FUNCTION_BLOCK SPLIT_AL_INTO_AQ (* this Function splits the 32 AQ (QUARTER) adapters from a AL (LWORD) *)
  (* Standard: 61499-2; Description: Copyright (c) 2026 Meisterschulen am Ostbahnhof SPDX-License-Identifier: EPL-2.0 *)
  (* Version 1.0, 2026-05-16, Franz Höpfinger, Meisterschulen am Ostbahnhof, initial API and implementation and/or initial documentation *)
  PACKAGE adapter::splitting;
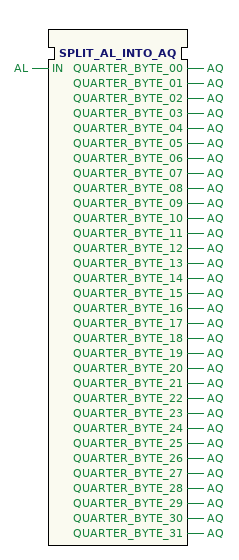
  SOCKETS
    IN : adapter::types::unidirectional::AL; (* LWORD Input *)
  END_SOCKETS
  PLUGS
    QUARTER_BYTE_00 : adapter::types::unidirectional::AQ; (* Quarter 0 *)
    QUARTER_BYTE_01 : adapter::types::unidirectional::AQ; (* Quarter 1 *)
    QUARTER_BYTE_02 : adapter::types::unidirectional::AQ; (* Quarter 2 *)
    QUARTER_BYTE_03 : adapter::types::unidirectional::AQ; (* Quarter 3 *)
    QUARTER_BYTE_04 : adapter::types::unidirectional::AQ; (* Quarter 4 *)
    QUARTER_BYTE_05 : adapter::types::unidirectional::AQ; (* Quarter 5 *)
    QUARTER_BYTE_06 : adapter::types::unidirectional::AQ; (* Quarter 6 *)
    QUARTER_BYTE_07 : adapter::types::unidirectional::AQ; (* Quarter 7 *)
    QUARTER_BYTE_08 : adapter::types::unidirectional::AQ; (* Quarter 8 *)
    QUARTER_BYTE_09 : adapter::types::unidirectional::AQ; (* Quarter 9 *)
    QUARTER_BYTE_10 : adapter::types::unidirectional::AQ; (* Quarter 10 *)
    QUARTER_BYTE_11 : adapter::types::unidirectional::AQ; (* Quarter 11 *)
    QUARTER_BYTE_12 : adapter::types::unidirectional::AQ; (* Quarter 12 *)
    QUARTER_BYTE_13 : adapter::types::unidirectional::AQ; (* Quarter 13 *)
    QUARTER_BYTE_14 : adapter::types::unidirectional::AQ; (* Quarter 14 *)
    QUARTER_BYTE_15 : adapter::types::unidirectional::AQ; (* Quarter 15 *)
    QUARTER_BYTE_16 : adapter::types::unidirectional::AQ; (* Quarter 16 *)
    QUARTER_BYTE_17 : adapter::types::unidirectional::AQ; (* Quarter 17 *)
    QUARTER_BYTE_18 : adapter::types::unidirectional::AQ; (* Quarter 18 *)
    QUARTER_BYTE_19 : adapter::types::unidirectional::AQ; (* Quarter 19 *)
    QUARTER_BYTE_20 : adapter::types::unidirectional::AQ; (* Quarter 20 *)
    QUARTER_BYTE_21 : adapter::types::unidirectional::AQ; (* Quarter 21 *)
    QUARTER_BYTE_22 : adapter::types::unidirectional::AQ; (* Quarter 22 *)
    QUARTER_BYTE_23 : adapter::types::unidirectional::AQ; (* Quarter 23 *)
    QUARTER_BYTE_24 : adapter::types::unidirectional::AQ; (* Quarter 24 *)
    QUARTER_BYTE_25 : adapter::types::unidirectional::AQ; (* Quarter 25 *)
    QUARTER_BYTE_26 : adapter::types::unidirectional::AQ; (* Quarter 26 *)
    QUARTER_BYTE_27 : adapter::types::unidirectional::AQ; (* Quarter 27 *)
    QUARTER_BYTE_28 : adapter::types::unidirectional::AQ; (* Quarter 28 *)
    QUARTER_BYTE_29 : adapter::types::unidirectional::AQ; (* Quarter 29 *)
    QUARTER_BYTE_30 : adapter::types::unidirectional::AQ; (* Quarter 30 *)
    QUARTER_BYTE_31 : adapter::types::unidirectional::AQ; (* Quarter 31 *)
  END_PLUGS
  FBS
    E_D_FF_ANY_00 : iec61499::events::E_D_FF_ANY;
    E_D_FF_ANY_01 : iec61499::events::E_D_FF_ANY;
    E_D_FF_ANY_02 : iec61499::events::E_D_FF_ANY;
    E_D_FF_ANY_03 : iec61499::events::E_D_FF_ANY;
    E_D_FF_ANY_04 : iec61499::events::E_D_FF_ANY;
    E_D_FF_ANY_05 : iec61499::events::E_D_FF_ANY;
    E_D_FF_ANY_06 : iec61499::events::E_D_FF_ANY;
    E_D_FF_ANY_07 : iec61499::events::E_D_FF_ANY;
    E_D_FF_ANY_08 : iec61499::events::E_D_FF_ANY;
    E_D_FF_ANY_09 : iec61499::events::E_D_FF_ANY;
    E_D_FF_ANY_10 : iec61499::events::E_D_FF_ANY;
    E_D_FF_ANY_11 : iec61499::events::E_D_FF_ANY;
    E_D_FF_ANY_12 : iec61499::events::E_D_FF_ANY;
    E_D_FF_ANY_13 : iec61499::events::E_D_FF_ANY;
    E_D_FF_ANY_14 : iec61499::events::E_D_FF_ANY;
    E_D_FF_ANY_15 : iec61499::events::E_D_FF_ANY;
    E_D_FF_ANY_16 : iec61499::events::E_D_FF_ANY;
    E_D_FF_ANY_17 : iec61499::events::E_D_FF_ANY;
    E_D_FF_ANY_18 : iec61499::events::E_D_FF_ANY;
    E_D_FF_ANY_19 : iec61499::events::E_D_FF_ANY;
    E_D_FF_ANY_20 : iec61499::events::E_D_FF_ANY;
    E_D_FF_ANY_21 : iec61499::events::E_D_FF_ANY;
    E_D_FF_ANY_22 : iec61499::events::E_D_FF_ANY;
    E_D_FF_ANY_23 : iec61499::events::E_D_FF_ANY;
    E_D_FF_ANY_24 : iec61499::events::E_D_FF_ANY;
    E_D_FF_ANY_25 : iec61499::events::E_D_FF_ANY;
    E_D_FF_ANY_26 : iec61499::events::E_D_FF_ANY;
    E_D_FF_ANY_27 : iec61499::events::E_D_FF_ANY;
    E_D_FF_ANY_28 : iec61499::events::E_D_FF_ANY;
    E_D_FF_ANY_29 : iec61499::events::E_D_FF_ANY;
    E_D_FF_ANY_30 : iec61499::events::E_D_FF_ANY;
    E_D_FF_ANY_31 : iec61499::events::E_D_FF_ANY;
    SPLIT_LWORD_INTO_QUARTERS : eclipse4diac::utils::splitting::SPLIT_LWORD_INTO_QUARTERS;
  END_FBS
  EVENT_CONNECTIONS
    IN.E1 TO SPLIT_LWORD_INTO_QUARTERS.REQ;
    SPLIT_LWORD_INTO_QUARTERS.CNF TO E_D_FF_ANY_00.CLK;
    SPLIT_LWORD_INTO_QUARTERS.CNF TO E_D_FF_ANY_01.CLK;
    SPLIT_LWORD_INTO_QUARTERS.CNF TO E_D_FF_ANY_02.CLK;
    SPLIT_LWORD_INTO_QUARTERS.CNF TO E_D_FF_ANY_03.CLK;
    SPLIT_LWORD_INTO_QUARTERS.CNF TO E_D_FF_ANY_04.CLK;
    SPLIT_LWORD_INTO_QUARTERS.CNF TO E_D_FF_ANY_05.CLK;
    SPLIT_LWORD_INTO_QUARTERS.CNF TO E_D_FF_ANY_06.CLK;
    SPLIT_LWORD_INTO_QUARTERS.CNF TO E_D_FF_ANY_07.CLK;
    SPLIT_LWORD_INTO_QUARTERS.CNF TO E_D_FF_ANY_08.CLK;
    SPLIT_LWORD_INTO_QUARTERS.CNF TO E_D_FF_ANY_09.CLK;
    SPLIT_LWORD_INTO_QUARTERS.CNF TO E_D_FF_ANY_10.CLK;
    SPLIT_LWORD_INTO_QUARTERS.CNF TO E_D_FF_ANY_11.CLK;
    SPLIT_LWORD_INTO_QUARTERS.CNF TO E_D_FF_ANY_12.CLK;
    SPLIT_LWORD_INTO_QUARTERS.CNF TO E_D_FF_ANY_13.CLK;
    SPLIT_LWORD_INTO_QUARTERS.CNF TO E_D_FF_ANY_14.CLK;
    SPLIT_LWORD_INTO_QUARTERS.CNF TO E_D_FF_ANY_15.CLK;
    SPLIT_LWORD_INTO_QUARTERS.CNF TO E_D_FF_ANY_16.CLK;
    SPLIT_LWORD_INTO_QUARTERS.CNF TO E_D_FF_ANY_17.CLK;
    SPLIT_LWORD_INTO_QUARTERS.CNF TO E_D_FF_ANY_18.CLK;
    SPLIT_LWORD_INTO_QUARTERS.CNF TO E_D_FF_ANY_19.CLK;
    SPLIT_LWORD_INTO_QUARTERS.CNF TO E_D_FF_ANY_20.CLK;
    SPLIT_LWORD_INTO_QUARTERS.CNF TO E_D_FF_ANY_21.CLK;
    SPLIT_LWORD_INTO_QUARTERS.CNF TO E_D_FF_ANY_22.CLK;
    SPLIT_LWORD_INTO_QUARTERS.CNF TO E_D_FF_ANY_23.CLK;
    SPLIT_LWORD_INTO_QUARTERS.CNF TO E_D_FF_ANY_24.CLK;
    SPLIT_LWORD_INTO_QUARTERS.CNF TO E_D_FF_ANY_25.CLK;
    SPLIT_LWORD_INTO_QUARTERS.CNF TO E_D_FF_ANY_26.CLK;
    SPLIT_LWORD_INTO_QUARTERS.CNF TO E_D_FF_ANY_27.CLK;
    SPLIT_LWORD_INTO_QUARTERS.CNF TO E_D_FF_ANY_28.CLK;
    SPLIT_LWORD_INTO_QUARTERS.CNF TO E_D_FF_ANY_29.CLK;
    SPLIT_LWORD_INTO_QUARTERS.CNF TO E_D_FF_ANY_30.CLK;
    SPLIT_LWORD_INTO_QUARTERS.CNF TO E_D_FF_ANY_31.CLK;
    E_D_FF_ANY_00.EO TO QUARTER_BYTE_00.E1;
    E_D_FF_ANY_01.EO TO QUARTER_BYTE_01.E1;
    E_D_FF_ANY_02.EO TO QUARTER_BYTE_02.E1;
    E_D_FF_ANY_03.EO TO QUARTER_BYTE_03.E1;
    E_D_FF_ANY_04.EO TO QUARTER_BYTE_04.E1;
    E_D_FF_ANY_05.EO TO QUARTER_BYTE_05.E1;
    E_D_FF_ANY_06.EO TO QUARTER_BYTE_06.E1;
    E_D_FF_ANY_07.EO TO QUARTER_BYTE_07.E1;
    E_D_FF_ANY_08.EO TO QUARTER_BYTE_08.E1;
    E_D_FF_ANY_09.EO TO QUARTER_BYTE_09.E1;
    E_D_FF_ANY_10.EO TO QUARTER_BYTE_10.E1;
    E_D_FF_ANY_11.EO TO QUARTER_BYTE_11.E1;
    E_D_FF_ANY_12.EO TO QUARTER_BYTE_12.E1;
    E_D_FF_ANY_13.EO TO QUARTER_BYTE_13.E1;
    E_D_FF_ANY_14.EO TO QUARTER_BYTE_14.E1;
    E_D_FF_ANY_15.EO TO QUARTER_BYTE_15.E1;
    E_D_FF_ANY_16.EO TO QUARTER_BYTE_16.E1;
    E_D_FF_ANY_17.EO TO QUARTER_BYTE_17.E1;
    E_D_FF_ANY_18.EO TO QUARTER_BYTE_18.E1;
    E_D_FF_ANY_19.EO TO QUARTER_BYTE_19.E1;
    E_D_FF_ANY_20.EO TO QUARTER_BYTE_20.E1;
    E_D_FF_ANY_21.EO TO QUARTER_BYTE_21.E1;
    E_D_FF_ANY_22.EO TO QUARTER_BYTE_22.E1;
    E_D_FF_ANY_23.EO TO QUARTER_BYTE_23.E1;
    E_D_FF_ANY_24.EO TO QUARTER_BYTE_24.E1;
    E_D_FF_ANY_25.EO TO QUARTER_BYTE_25.E1;
    E_D_FF_ANY_26.EO TO QUARTER_BYTE_26.E1;
    E_D_FF_ANY_27.EO TO QUARTER_BYTE_27.E1;
    E_D_FF_ANY_28.EO TO QUARTER_BYTE_28.E1;
    E_D_FF_ANY_29.EO TO QUARTER_BYTE_29.E1;
    E_D_FF_ANY_30.EO TO QUARTER_BYTE_30.E1;
    E_D_FF_ANY_31.EO TO QUARTER_BYTE_31.E1;
  END_CONNECTIONS
  DATA_CONNECTIONS
    IN.D1 TO SPLIT_LWORD_INTO_QUARTERS.IN;
    SPLIT_LWORD_INTO_QUARTERS.QUARTER_BYTE_31 TO E_D_FF_ANY_31.D;
    SPLIT_LWORD_INTO_QUARTERS.QUARTER_BYTE_30 TO E_D_FF_ANY_30.D;
    SPLIT_LWORD_INTO_QUARTERS.QUARTER_BYTE_29 TO E_D_FF_ANY_29.D;
    SPLIT_LWORD_INTO_QUARTERS.QUARTER_BYTE_28 TO E_D_FF_ANY_28.D;
    SPLIT_LWORD_INTO_QUARTERS.QUARTER_BYTE_27 TO E_D_FF_ANY_27.D;
    SPLIT_LWORD_INTO_QUARTERS.QUARTER_BYTE_26 TO E_D_FF_ANY_26.D;
    SPLIT_LWORD_INTO_QUARTERS.QUARTER_BYTE_25 TO E_D_FF_ANY_25.D;
    SPLIT_LWORD_INTO_QUARTERS.QUARTER_BYTE_24 TO E_D_FF_ANY_24.D;
    SPLIT_LWORD_INTO_QUARTERS.QUARTER_BYTE_23 TO E_D_FF_ANY_23.D;
    SPLIT_LWORD_INTO_QUARTERS.QUARTER_BYTE_22 TO E_D_FF_ANY_22.D;
    SPLIT_LWORD_INTO_QUARTERS.QUARTER_BYTE_21 TO E_D_FF_ANY_21.D;
    SPLIT_LWORD_INTO_QUARTERS.QUARTER_BYTE_20 TO E_D_FF_ANY_20.D;
    SPLIT_LWORD_INTO_QUARTERS.QUARTER_BYTE_19 TO E_D_FF_ANY_19.D;
    SPLIT_LWORD_INTO_QUARTERS.QUARTER_BYTE_18 TO E_D_FF_ANY_18.D;
    SPLIT_LWORD_INTO_QUARTERS.QUARTER_BYTE_17 TO E_D_FF_ANY_17.D;
    SPLIT_LWORD_INTO_QUARTERS.QUARTER_BYTE_16 TO E_D_FF_ANY_16.D;
    SPLIT_LWORD_INTO_QUARTERS.QUARTER_BYTE_15 TO E_D_FF_ANY_15.D;
    SPLIT_LWORD_INTO_QUARTERS.QUARTER_BYTE_14 TO E_D_FF_ANY_14.D;
    SPLIT_LWORD_INTO_QUARTERS.QUARTER_BYTE_13 TO E_D_FF_ANY_13.D;
    SPLIT_LWORD_INTO_QUARTERS.QUARTER_BYTE_12 TO E_D_FF_ANY_12.D;
    SPLIT_LWORD_INTO_QUARTERS.QUARTER_BYTE_11 TO E_D_FF_ANY_11.D;
    SPLIT_LWORD_INTO_QUARTERS.QUARTER_BYTE_10 TO E_D_FF_ANY_10.D;
    SPLIT_LWORD_INTO_QUARTERS.QUARTER_BYTE_09 TO E_D_FF_ANY_09.D;
    SPLIT_LWORD_INTO_QUARTERS.QUARTER_BYTE_08 TO E_D_FF_ANY_08.D;
    SPLIT_LWORD_INTO_QUARTERS.QUARTER_BYTE_07 TO E_D_FF_ANY_07.D;
    SPLIT_LWORD_INTO_QUARTERS.QUARTER_BYTE_06 TO E_D_FF_ANY_06.D;
    SPLIT_LWORD_INTO_QUARTERS.QUARTER_BYTE_05 TO E_D_FF_ANY_05.D;
    SPLIT_LWORD_INTO_QUARTERS.QUARTER_BYTE_04 TO E_D_FF_ANY_04.D;
    SPLIT_LWORD_INTO_QUARTERS.QUARTER_BYTE_03 TO E_D_FF_ANY_03.D;
    SPLIT_LWORD_INTO_QUARTERS.QUARTER_BYTE_02 TO E_D_FF_ANY_02.D;
    SPLIT_LWORD_INTO_QUARTERS.QUARTER_BYTE_01 TO E_D_FF_ANY_01.D;
    SPLIT_LWORD_INTO_QUARTERS.QUARTER_BYTE_00 TO E_D_FF_ANY_00.D;
    E_D_FF_ANY_00.Q TO QUARTER_BYTE_00.D1;
    E_D_FF_ANY_01.Q TO QUARTER_BYTE_01.D1;
    E_D_FF_ANY_02.Q TO QUARTER_BYTE_02.D1;
    E_D_FF_ANY_03.Q TO QUARTER_BYTE_03.D1;
    E_D_FF_ANY_04.Q TO QUARTER_BYTE_04.D1;
    E_D_FF_ANY_05.Q TO QUARTER_BYTE_05.D1;
    E_D_FF_ANY_06.Q TO QUARTER_BYTE_06.D1;
    E_D_FF_ANY_07.Q TO QUARTER_BYTE_07.D1;
    E_D_FF_ANY_08.Q TO QUARTER_BYTE_08.D1;
    E_D_FF_ANY_09.Q TO QUARTER_BYTE_09.D1;
    E_D_FF_ANY_10.Q TO QUARTER_BYTE_10.D1;
    E_D_FF_ANY_11.Q TO QUARTER_BYTE_11.D1;
    E_D_FF_ANY_12.Q TO QUARTER_BYTE_12.D1;
    E_D_FF_ANY_13.Q TO QUARTER_BYTE_13.D1;
    E_D_FF_ANY_14.Q TO QUARTER_BYTE_14.D1;
    E_D_FF_ANY_15.Q TO QUARTER_BYTE_15.D1;
    E_D_FF_ANY_16.Q TO QUARTER_BYTE_16.D1;
    E_D_FF_ANY_17.Q TO QUARTER_BYTE_17.D1;
    E_D_FF_ANY_18.Q TO QUARTER_BYTE_18.D1;
    E_D_FF_ANY_19.Q TO QUARTER_BYTE_19.D1;
    E_D_FF_ANY_20.Q TO QUARTER_BYTE_20.D1;
    E_D_FF_ANY_21.Q TO QUARTER_BYTE_21.D1;
    E_D_FF_ANY_22.Q TO QUARTER_BYTE_22.D1;
    E_D_FF_ANY_23.Q TO QUARTER_BYTE_23.D1;
    E_D_FF_ANY_24.Q TO QUARTER_BYTE_24.D1;
    E_D_FF_ANY_25.Q TO QUARTER_BYTE_25.D1;
    E_D_FF_ANY_26.Q TO QUARTER_BYTE_26.D1;
    E_D_FF_ANY_27.Q TO QUARTER_BYTE_27.D1;
    E_D_FF_ANY_28.Q TO QUARTER_BYTE_28.D1;
    E_D_FF_ANY_29.Q TO QUARTER_BYTE_29.D1;
    E_D_FF_ANY_30.Q TO QUARTER_BYTE_30.D1;
    E_D_FF_ANY_31.Q TO QUARTER_BYTE_31.D1;
  END_CONNECTIONS
END_FUNCTION_BLOCK
